(* IEC 61131-3 sources: UniTest/iecUniTest_br/Library_tests/main, 1 file *)

(* ---- main.st ---- *)
PROGRAM _CYCLIC
    (*https://github.com/tkucic/iecUniTest/blob/main/docs/docs/ns/Library_tests/prg/main.md*)
    testReporter(Results:=gResults);
END_PROGRAM
